// TIA Portal V20 export
TYPE "zm_LOGSOperationData2"
// stored: Access Published
   STRUCT
      ReachedtoCamearaPos : Bool;
      ReachedtoLoadPos : Bool;
      LoaderClamped : Bool;
      LoaderUnclamped : Bool;
      LoadComplete : Bool;
   END_STRUCT;
END_TYPE
